% RSLogix 500 project Project_7.RSS, saved by version 8.30.00.16 %
PROJECT "UNTITLED"    % processor: Bul.1763 MicroLogix 1100 Series B %

PROGRAM FILES
  LAD 2   4 rungs
  LAD 3 "CALIBRATIO"  8 rungs
  LAD 4 "IO"  8 rungs

DATA FILES
  O0 OUTPUT  9 elements
  I1 INPUT  16 elements
  S2 STATUS  66 elements
  B3 BINARY  1 elements
  T4 TIMER  3 elements
  C5 COUNTER  2 elements
  R6 CONTROL  1 elements
  N7 INTEGER  10 elements
  F8 FLOAT  9 elements

LADDER 2
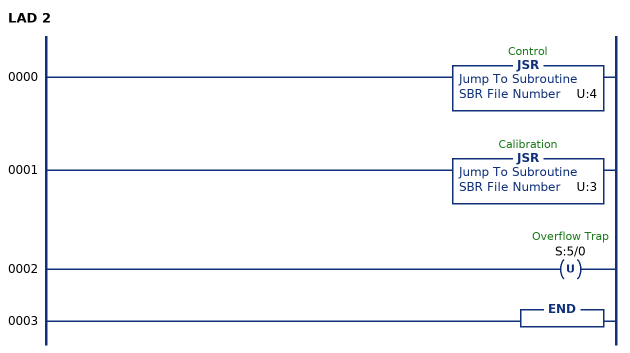
% Rung: 0 %
SOR JSR U:4 EOR
%   U:4  "Control" %
% Rung: 1 %
SOR JSR U:3 EOR
%   U:3  "Calibration" %
% Rung: 2 %
SOR OTU S:5/0 EOR
%   S:5/0  "Overflow Trap" %
% Rung: 3 %
SOR END EOR

LADDER 3 "CALIBRATIO"
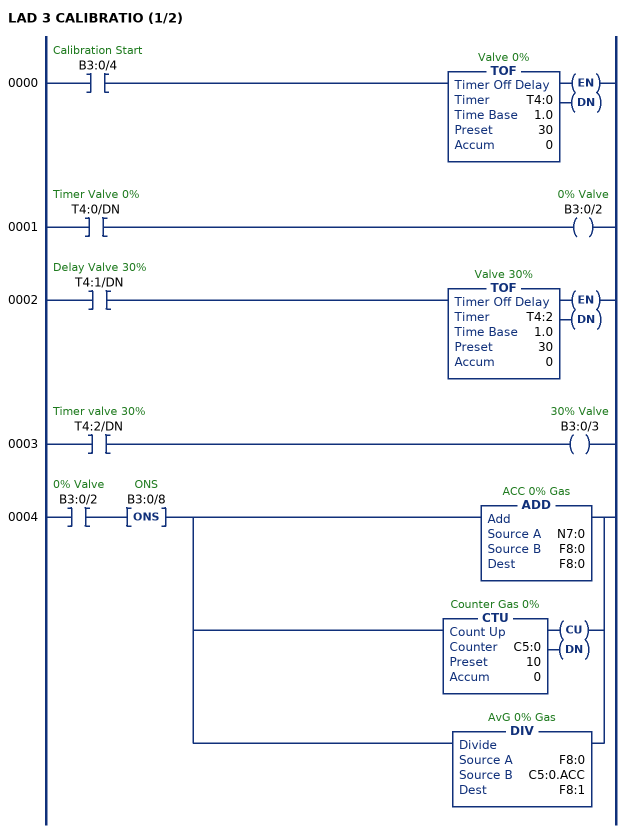
% Rung: 0 %
SOR XIC B3:0/4 TOF T4:0 1.0 30 0 EOR
%   B3:0/4  "Calibration Start" %
%   T4:0  "Valve 0%" %
% Rung: 1 %
SOR XIC T4:0/DN OTE B3:0/2 EOR
%   T4:0/DN  "Timer Valve 0%" %
%   B3:0/2  "0% Valve" %
% Rung: 2 %
SOR XIC T4:1/DN TOF T4:2 1.0 30 0 EOR
%   T4:1/DN  "Delay Valve 30%" %
%   T4:2  "Valve 30%" %
% Rung: 3 %
SOR XIC T4:2/DN OTE B3:0/3 EOR
%   T4:2/DN  "Timer valve 30%" %
%   B3:0/3  "30% Valve" %
% Rung: 4 %
SOR XIC B3:0/2 ONS B3:0/8 BST ADD N7:0 F8:0 F8:0 NXB CTU C5:0 10 0 NXB DIV F8:0 C5:0.ACC F8:1 BND EOR
%   B3:0/2  "0% Valve" %
%   B3:0/8  "ONS" %
%   N7:0  "O2 Sensor Input" %
%   F8:0  "ACC 0% Gas" %
%   C5:0  "Counter Gas 0%" %
%   C5:0.ACC  "Cunter Gas 0%" %
%   F8:1  "AvG 0% Gas" %

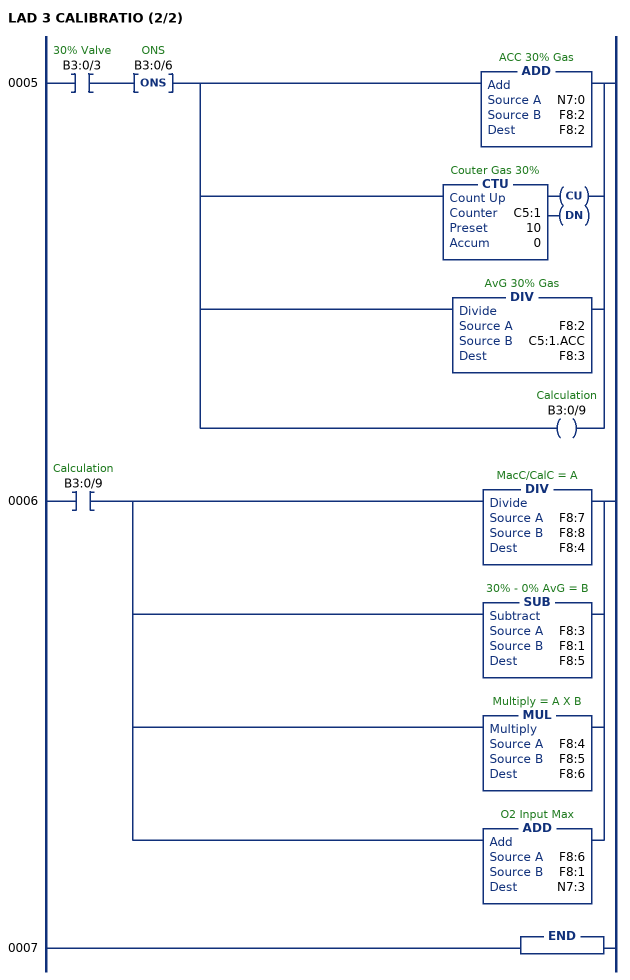
% Rung: 5 %
SOR XIC B3:0/3 ONS B3:0/6 BST ADD N7:0 F8:2 F8:2 NXB CTU C5:1 10 0 NXB DIV F8:2 C5:1.ACC F8:3 NXB OTE B3:0/9 BND EOR
%   B3:0/3  "30% Valve" %
%   B3:0/6  "ONS" %
%   N7:0  "O2 Sensor Input" %
%   F8:2  "ACC 30% Gas" %
%   C5:1  "Couter Gas 30%" %
%   C5:1.ACC  "Counter Gas 30%" %
%   F8:3  "AvG 30% Gas" %
%   B3:0/9  "Calculation" %
% Rung: 6 %
SOR XIC B3:0/9 BST DIV F8:7 F8:8 F8:4 NXB SUB F8:3 F8:1 F8:5 NXB MUL F8:4 F8:5 F8:6 NXB ADD F8:6 F8:1 N7:3 BND EOR
%   B3:0/9  "Calculation" %
%   F8:7  "40 % Gas" %
%   F8:8  "30% Gas" %
%   F8:4  "MacC/CalC = A" %
%   F8:3  "AvG 30% Gas" %
%   F8:1  "AvG 0% Gas" %
%   F8:5  "30% - 0% AvG = B" %
%   F8:6  "Multiply = A X B" %
%   N7:3  "O2 Input Max" %
% Rung: 7 %
SOR END EOR

LADDER 4 "IO"
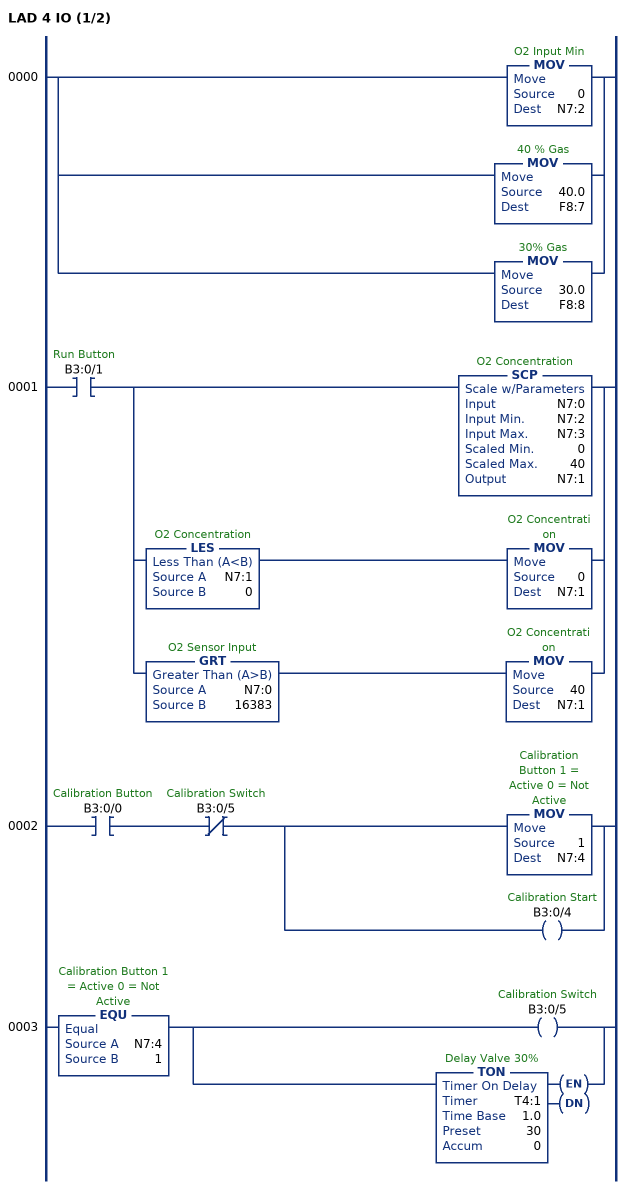
% Rung: 0 %
SOR BST MOV 0 N7:2 NXB MOV 40.0 F8:7 NXB MOV 30.0 F8:8 BND EOR
%   N7:2  "O2 Input Min" %
%   F8:7  "40 % Gas" %
%   F8:8  "30% Gas" %
% Rung: 1 %
SOR XIC B3:0/1 BST SCP N7:0 N7:2 N7:3 0 40 N7:1 NXB LES N7:1 0 MOV 0 N7:1 NXB GRT N7:0 16383 MOV 40 N7:1 BND EOR
%   B3:0/1  "Run Button" %
%   N7:0  "O2 Sensor Input" %
%   N7:2  "O2 Input Min" %
%   N7:3  "O2 Input Max" %
%   N7:1  "O2 Concentration" %
% Rung: 2 %
SOR XIC B3:0/0 XIO B3:0/5 BST MOV 1 N7:4 NXB OTE B3:0/4 BND EOR
%   B3:0/0  "Calibration Button" %
%   B3:0/5  "Calibration Switch" %
%   N7:4  "Calibration Button 1 = Active 0 = Not Active" %
%   B3:0/4  "Calibration Start" %
% Rung: 3 %
SOR EQU N7:4 1 BST OTE B3:0/5 NXB TON T4:1 1.0 30 0 BND EOR
%   N7:4  "Calibration Button 1 = Active 0 = Not Active" %
%   B3:0/5  "Calibration Switch" %
%   T4:1  "Delay Valve 30%" %

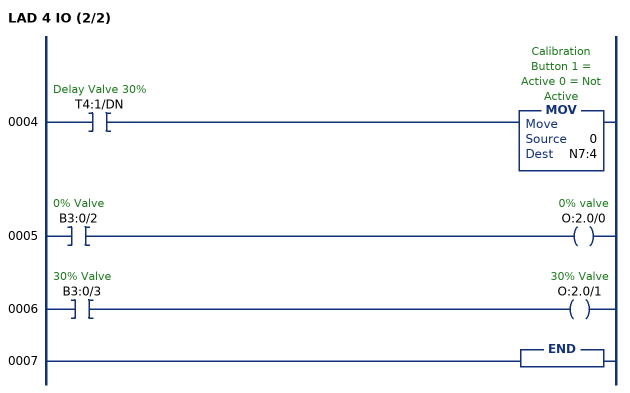
% Rung: 4 %
SOR XIC T4:1/DN MOV 0 N7:4 EOR
%   T4:1/DN  "Delay Valve 30%" %
%   N7:4  "Calibration Button 1 = Active 0 = Not Active" %
% Rung: 5 %
SOR XIC B3:0/2 OTE O:2.0/0 EOR
%   B3:0/2  "0% Valve" %
%   O:2.0/0  "0% valve" %
% Rung: 6 %
SOR XIC B3:0/3 OTE O:2.0/1 EOR
%   B3:0/3  "30% Valve" %
%   O:2.0/1  "30% Valve" %
% Rung: 7 %
SOR END EOR

OTHER DOCUMENTED ADDRESSES
  B3:0/7  "Gate Constant 0"
  B3:7  "Gate Constant 0"
  I:3  "Gas Sensor"
  I:3.0/0  "Sensor Gas"
  I:3.0/1  "Gas Sensor"
  N7:5  "ACC Gas 30%"
  N7:6  "ACC Gas 30%"
  N7:7  "ACC Gas 30%"
  N7:8  "Acc Gas 30%"
  N7:9  "Gate Constant 0 1 = Active 0 = Not Active"
  T4:0/1  "Timer Reset Calibration"

DATA TABLE (non-zero values as saved)
DATA T4
% .PRE .ACC %
% T4:0 % 30 0
% T4:1 % 30 0
% T4:2 % 30 0
DATA C5
% .PRE .ACC %
% C5:0 % 10 0
% C5:1 % 10 0
DATA N7
% N7:0 % 8192 0 0 16383 0 0 0 0 0 0
